PROGRAM IO_Mapping
VAR
	BLINK_500msOn_500MsOff	: Blink;
END_VAR

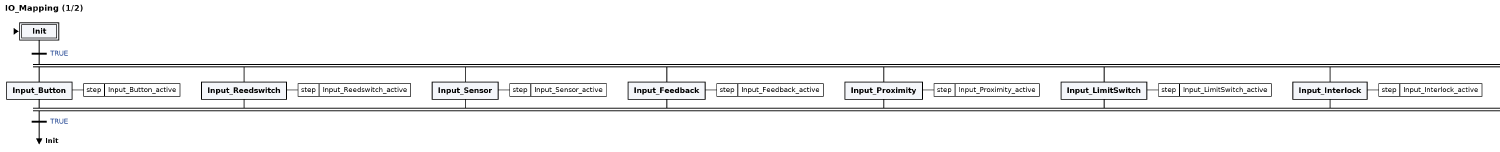
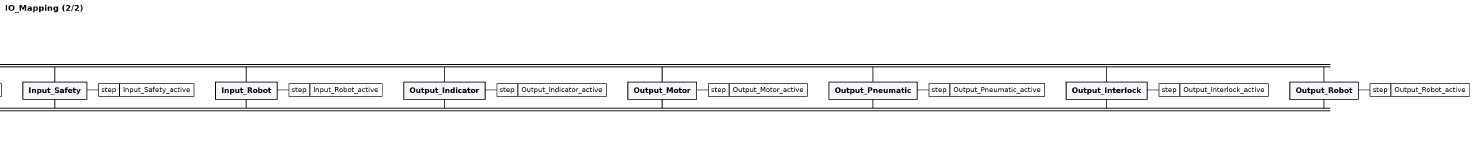
INITIAL_STEP Init:
END_STEP
TRANSITION FROM Init TO (Input_Button, Input_Reedswitch, Input_Sensor, Input_Feedback, Input_Proximity, Input_LimitSwitch, Input_Interlock, Input_Safety, Input_Robot, Output_Indicator, Output_Motor, Output_Pneumatic, Output_Interlock, Output_Robot)
    := TRUE;
END_TRANSITION
STEP Input_Button:
    Input_Button_active(N);  // step action
END_STEP
STEP Input_Reedswitch:
    Input_Reedswitch_active(N);  // step action
END_STEP
STEP Input_Sensor:
    Input_Sensor_active(N);  // step action
END_STEP
STEP Input_Feedback:
    Input_Feedback_active(N);  // step action
END_STEP
STEP Input_Proximity:
    Input_Proximity_active(N);  // step action
END_STEP
STEP Input_LimitSwitch:
    Input_LimitSwitch_active(N);  // step action
END_STEP
STEP Input_Interlock:
    Input_Interlock_active(N);  // step action
END_STEP
STEP Input_Safety:
    Input_Safety_active(N);  // step action
END_STEP
STEP Input_Robot:
    Input_Robot_active(N);  // step action
END_STEP
STEP Output_Indicator:
    Output_Indicator_active(N);  // step action
END_STEP
STEP Output_Motor:
    Output_Motor_active(N);  // step action
END_STEP
STEP Output_Pneumatic:
    Output_Pneumatic_active(N);  // step action
END_STEP
STEP Output_Interlock:
    Output_Interlock_active(N);  // step action
END_STEP
STEP Output_Robot:
    Output_Robot_active(N);  // step action
END_STEP
TRANSITION FROM (Input_Button, Input_Reedswitch, Input_Sensor, Input_Feedback, Input_Proximity, Input_LimitSwitch, Input_Interlock, Input_Safety, Input_Robot, Output_Indicator, Output_Motor, Output_Pneumatic, Output_Interlock, Output_Robot) TO Init
    := TRUE;
END_TRANSITION

ACTION Input_Button_active:
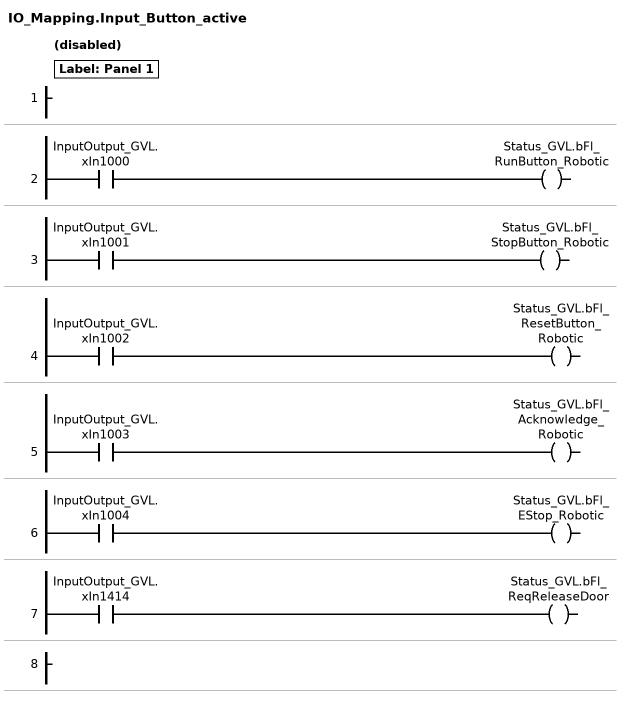
// NETWORK 1 (disabled)
// label: Label: Panel 1

// NETWORK 2
Status_GVL.bFl_RunButton_Robotic := InputOutput_GVL.xIn1000;

// NETWORK 3
Status_GVL.bFl_StopButton_Robotic := InputOutput_GVL.xIn1001;

// NETWORK 4
Status_GVL.bFl_ResetButton_Robotic := InputOutput_GVL.xIn1002;

// NETWORK 5
Status_GVL.bFl_Acknowledge_Robotic := InputOutput_GVL.xIn1003;

// NETWORK 6
Status_GVL.bFl_EStop_Robotic := InputOutput_GVL.xIn1004;

// NETWORK 7
Status_GVL.bFl_ReqReleaseDoor := InputOutput_GVL.xIn1414;

// NETWORK 8
END_ACTION

ACTION Input_Feedback_active:
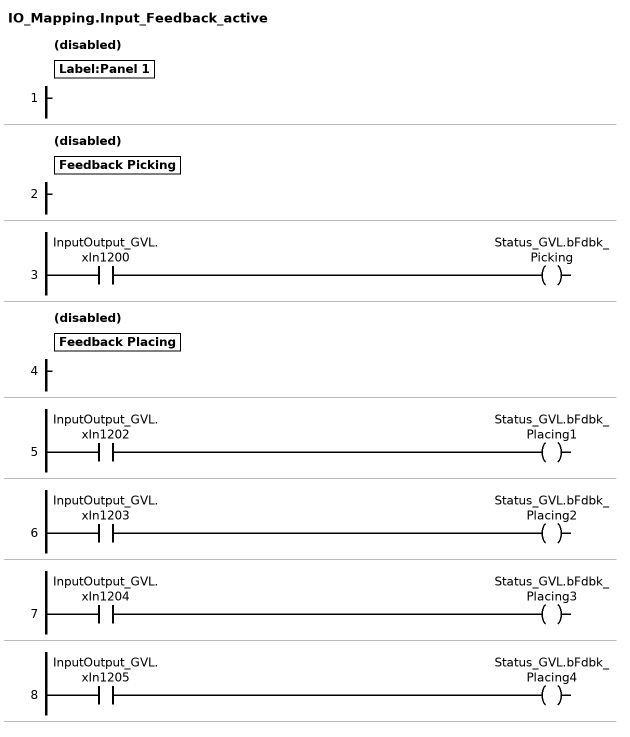
// NETWORK 1 (disabled)
// label: Label:Panel 1

// NETWORK 2 (disabled)
// label: Feedback Picking

// NETWORK 3
Status_GVL.bFdbk_Picking := InputOutput_GVL.xIn1200;

// NETWORK 4 (disabled)
// label: Feedback Placing

// NETWORK 5
Status_GVL.bFdbk_Placing1 := InputOutput_GVL.xIn1202;

// NETWORK 6
Status_GVL.bFdbk_Placing2 := InputOutput_GVL.xIn1203;

// NETWORK 7
Status_GVL.bFdbk_Placing3 := InputOutput_GVL.xIn1204;

// NETWORK 8
Status_GVL.bFdbk_Placing4 := InputOutput_GVL.xIn1205;
END_ACTION

ACTION Input_Interlock_active:
// NETWORK 1
END_ACTION

ACTION Input_LimitSwitch_active:
// NETWORK 1
END_ACTION

ACTION Input_Proximity_active:
// NETWORK 1 (disabled)
// label: Proximity

// NETWORK 2
END_ACTION

ACTION Input_Reedswitch_active:
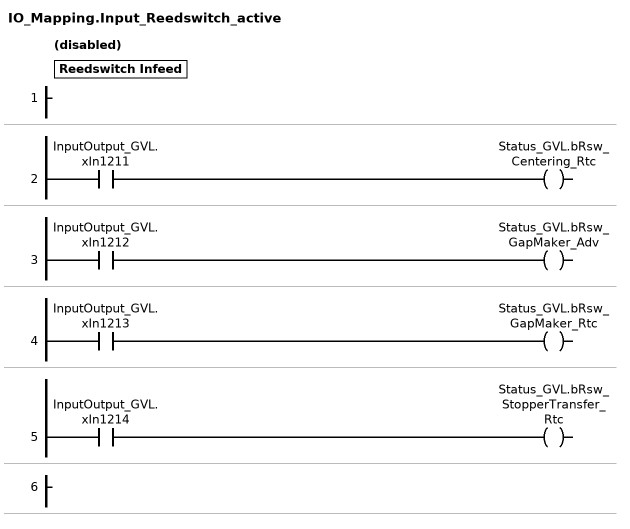
// NETWORK 1 (disabled)
// label: Reedswitch Infeed

// NETWORK 2
Status_GVL.bRsw_Centering_Rtc := InputOutput_GVL.xIn1211;

// NETWORK 3
Status_GVL.bRsw_GapMaker_Adv := InputOutput_GVL.xIn1212;

// NETWORK 4
Status_GVL.bRsw_GapMaker_Rtc := InputOutput_GVL.xIn1213;

// NETWORK 5
Status_GVL.bRsw_StopperTransfer_Rtc := InputOutput_GVL.xIn1214;

// NETWORK 6
END_ACTION

ACTION Input_Robot_active:
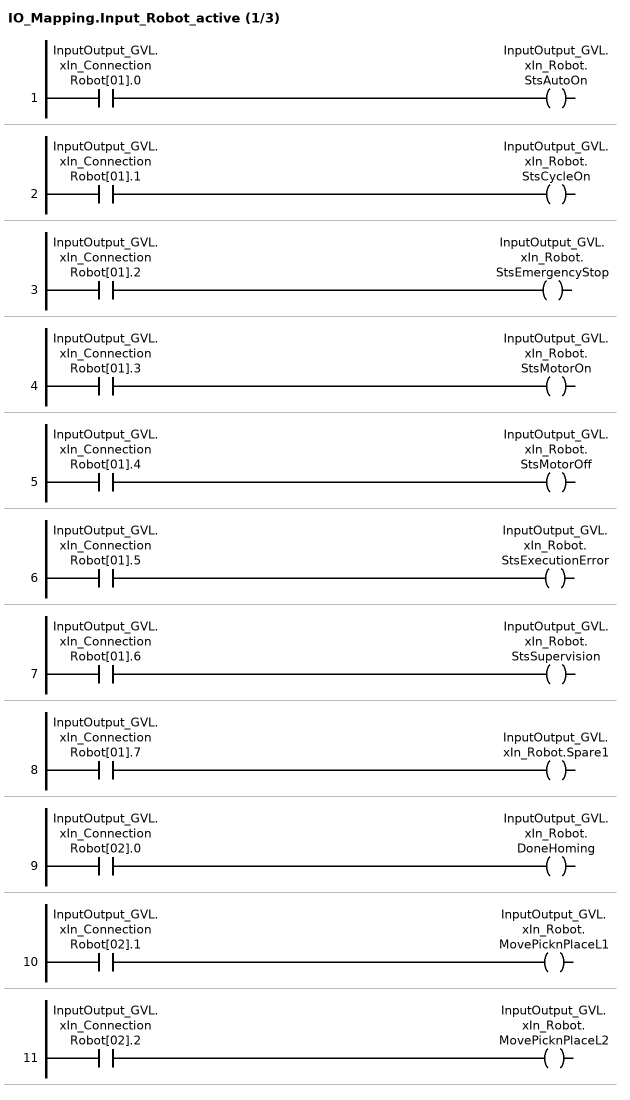
// NETWORK 1
InputOutput_GVL.xIn_Robot.StsAutoOn := InputOutput_GVL.xIn_ConnectionRobot[01].0;

// NETWORK 2
InputOutput_GVL.xIn_Robot.StsCycleOn := InputOutput_GVL.xIn_ConnectionRobot[01].1;

// NETWORK 3
InputOutput_GVL.xIn_Robot.StsEmergencyStop := InputOutput_GVL.xIn_ConnectionRobot[01].2;

// NETWORK 4
InputOutput_GVL.xIn_Robot.StsMotorOn := InputOutput_GVL.xIn_ConnectionRobot[01].3;

// NETWORK 5
InputOutput_GVL.xIn_Robot.StsMotorOff := InputOutput_GVL.xIn_ConnectionRobot[01].4;

// NETWORK 6
InputOutput_GVL.xIn_Robot.StsExecutionError := InputOutput_GVL.xIn_ConnectionRobot[01].5;

// NETWORK 7
InputOutput_GVL.xIn_Robot.StsSupervision := InputOutput_GVL.xIn_ConnectionRobot[01].6;

// NETWORK 8
InputOutput_GVL.xIn_Robot.Spare1 := InputOutput_GVL.xIn_ConnectionRobot[01].7;

// NETWORK 9
InputOutput_GVL.xIn_Robot.DoneHoming := InputOutput_GVL.xIn_ConnectionRobot[02].0;

// NETWORK 10
InputOutput_GVL.xIn_Robot.MovePicknPlaceL1 := InputOutput_GVL.xIn_ConnectionRobot[02].1;

// NETWORK 11
InputOutput_GVL.xIn_Robot.MovePicknPlaceL2 := InputOutput_GVL.xIn_ConnectionRobot[02].2;

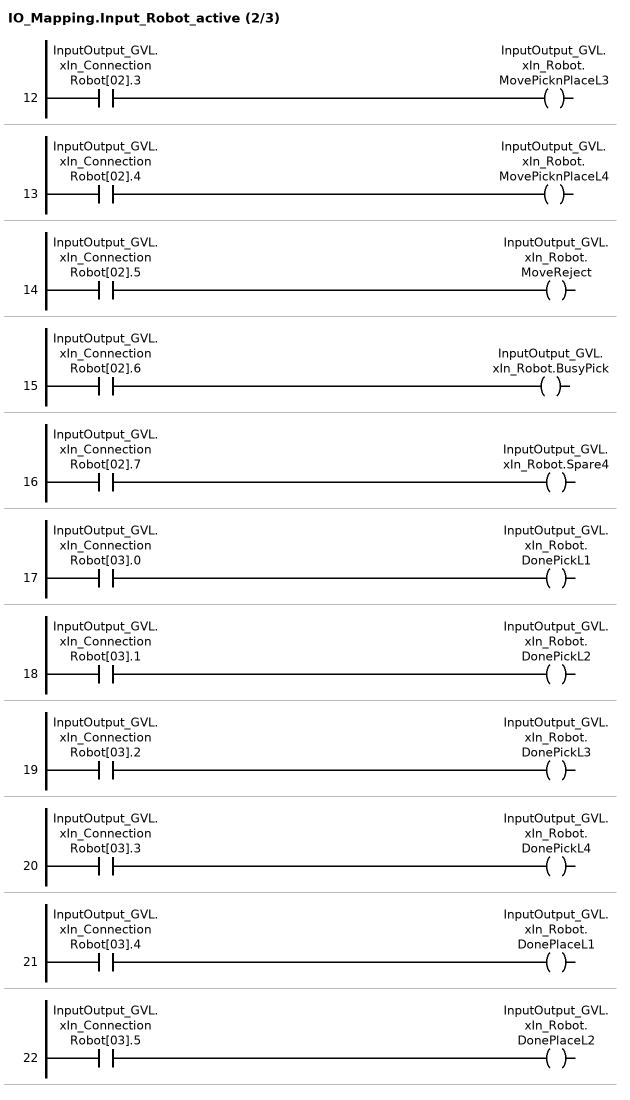
// NETWORK 12
InputOutput_GVL.xIn_Robot.MovePicknPlaceL3 := InputOutput_GVL.xIn_ConnectionRobot[02].3;

// NETWORK 13
InputOutput_GVL.xIn_Robot.MovePicknPlaceL4 := InputOutput_GVL.xIn_ConnectionRobot[02].4;

// NETWORK 14
InputOutput_GVL.xIn_Robot.MoveReject := InputOutput_GVL.xIn_ConnectionRobot[02].5;

// NETWORK 15
InputOutput_GVL.xIn_Robot.BusyPick := InputOutput_GVL.xIn_ConnectionRobot[02].6;

// NETWORK 16
InputOutput_GVL.xIn_Robot.Spare4 := InputOutput_GVL.xIn_ConnectionRobot[02].7;

// NETWORK 17
InputOutput_GVL.xIn_Robot.DonePickL1 := InputOutput_GVL.xIn_ConnectionRobot[03].0;

// NETWORK 18
InputOutput_GVL.xIn_Robot.DonePickL2 := InputOutput_GVL.xIn_ConnectionRobot[03].1;

// NETWORK 19
InputOutput_GVL.xIn_Robot.DonePickL3 := InputOutput_GVL.xIn_ConnectionRobot[03].2;

// NETWORK 20
InputOutput_GVL.xIn_Robot.DonePickL4 := InputOutput_GVL.xIn_ConnectionRobot[03].3;

// NETWORK 21
InputOutput_GVL.xIn_Robot.DonePlaceL1 := InputOutput_GVL.xIn_ConnectionRobot[03].4;

// NETWORK 22
InputOutput_GVL.xIn_Robot.DonePlaceL2 := InputOutput_GVL.xIn_ConnectionRobot[03].5;

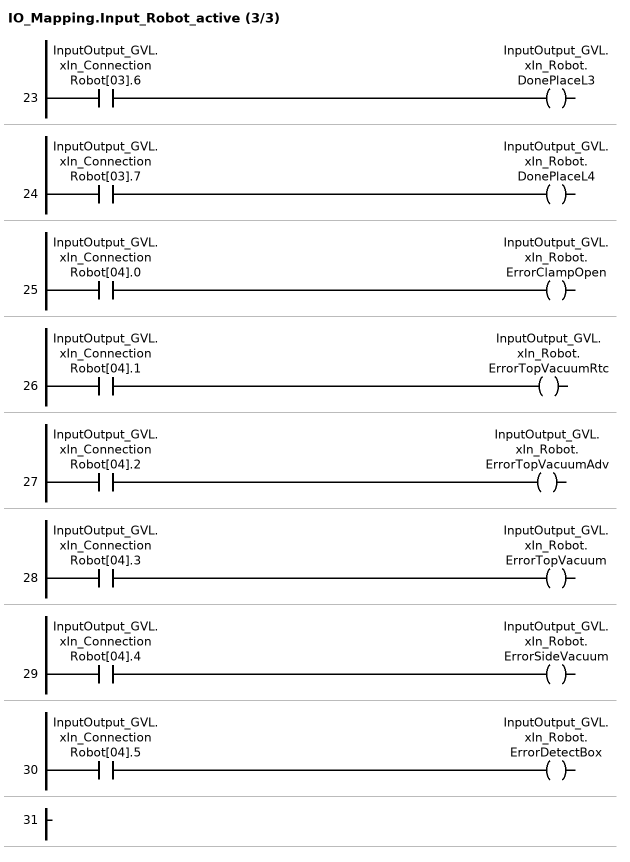
// NETWORK 23
InputOutput_GVL.xIn_Robot.DonePlaceL3 := InputOutput_GVL.xIn_ConnectionRobot[03].6;

// NETWORK 24
InputOutput_GVL.xIn_Robot.DonePlaceL4 := InputOutput_GVL.xIn_ConnectionRobot[03].7;

// NETWORK 25
InputOutput_GVL.xIn_Robot.ErrorClampOpen := InputOutput_GVL.xIn_ConnectionRobot[04].0;

// NETWORK 26
InputOutput_GVL.xIn_Robot.ErrorTopVacuumRtc := InputOutput_GVL.xIn_ConnectionRobot[04].1;

// NETWORK 27
InputOutput_GVL.xIn_Robot.ErrorTopVacuumAdv := InputOutput_GVL.xIn_ConnectionRobot[04].2;

// NETWORK 28
InputOutput_GVL.xIn_Robot.ErrorTopVacuum := InputOutput_GVL.xIn_ConnectionRobot[04].3;

// NETWORK 29
InputOutput_GVL.xIn_Robot.ErrorSideVacuum := InputOutput_GVL.xIn_ConnectionRobot[04].4;

// NETWORK 30
InputOutput_GVL.xIn_Robot.ErrorDetectBox := InputOutput_GVL.xIn_ConnectionRobot[04].5;

// NETWORK 31
END_ACTION

ACTION Input_Safety_active:
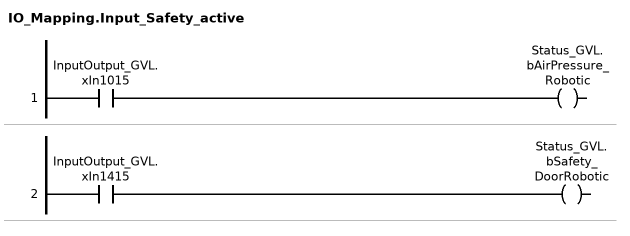
// NETWORK 1
Status_GVL.bAirPressure_Robotic := InputOutput_GVL.xIn1015;

// NETWORK 2
Status_GVL.bSafety_DoorRobotic := InputOutput_GVL.xIn1415;
END_ACTION

ACTION Input_Sensor_active:
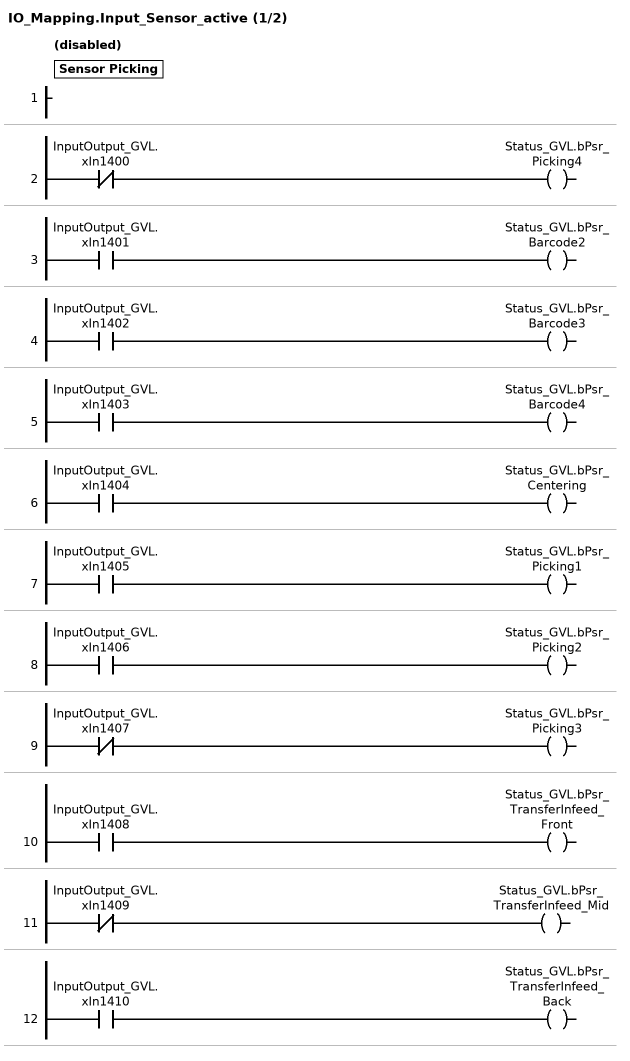
// NETWORK 1 (disabled)
// label: Sensor Picking

// NETWORK 2
Status_GVL.bPsr_Picking4 := NOT InputOutput_GVL.xIn1400;

// NETWORK 3
Status_GVL.bPsr_Barcode2 := InputOutput_GVL.xIn1401;

// NETWORK 4
Status_GVL.bPsr_Barcode3 := InputOutput_GVL.xIn1402;

// NETWORK 5
Status_GVL.bPsr_Barcode4 := InputOutput_GVL.xIn1403;

// NETWORK 6
Status_GVL.bPsr_Centering := InputOutput_GVL.xIn1404;

// NETWORK 7
Status_GVL.bPsr_Picking1 := InputOutput_GVL.xIn1405;

// NETWORK 8
Status_GVL.bPsr_Picking2 := InputOutput_GVL.xIn1406;

// NETWORK 9
Status_GVL.bPsr_Picking3 := NOT InputOutput_GVL.xIn1407;

// NETWORK 10
Status_GVL.bPsr_TransferInfeed_Front := InputOutput_GVL.xIn1408;

// NETWORK 11
Status_GVL.bPsr_TransferInfeed_Mid := NOT InputOutput_GVL.xIn1409;

// NETWORK 12
Status_GVL.bPsr_TransferInfeed_Back := InputOutput_GVL.xIn1410;

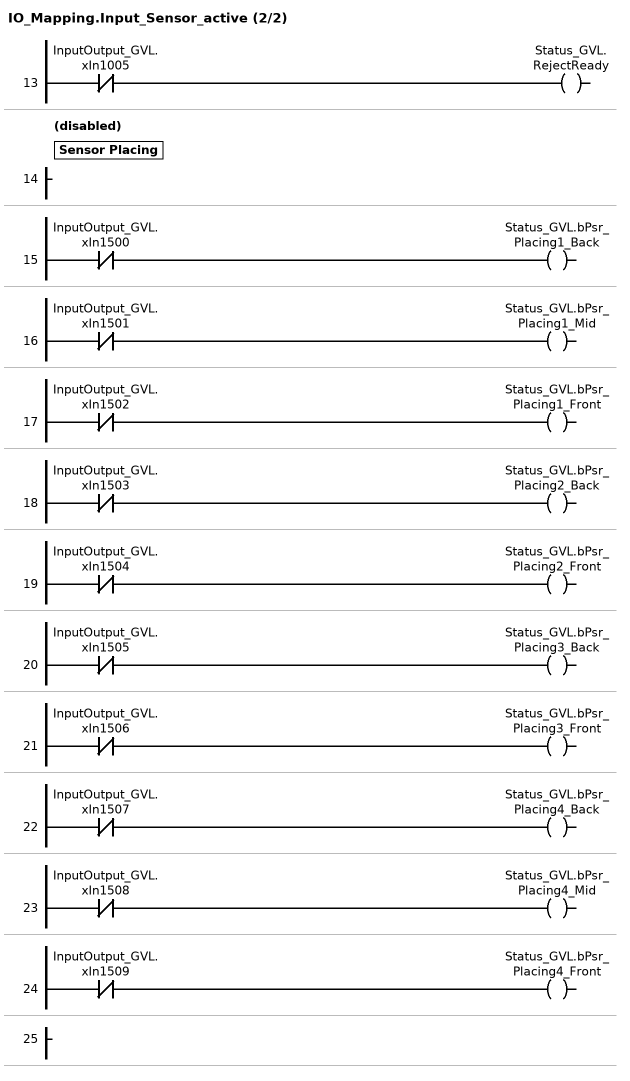
// NETWORK 13
Status_GVL.RejectReady := NOT InputOutput_GVL.xIn1005;

// NETWORK 14 (disabled)
// label: Sensor Placing

// NETWORK 15
Status_GVL.bPsr_Placing1_Back := NOT InputOutput_GVL.xIn1500;

// NETWORK 16
Status_GVL.bPsr_Placing1_Mid := NOT InputOutput_GVL.xIn1501;

// NETWORK 17
Status_GVL.bPsr_Placing1_Front := NOT InputOutput_GVL.xIn1502;

// NETWORK 18
Status_GVL.bPsr_Placing2_Back := NOT InputOutput_GVL.xIn1503;

// NETWORK 19
Status_GVL.bPsr_Placing2_Front := NOT InputOutput_GVL.xIn1504;

// NETWORK 20
Status_GVL.bPsr_Placing3_Back := NOT InputOutput_GVL.xIn1505;

// NETWORK 21
Status_GVL.bPsr_Placing3_Front := NOT InputOutput_GVL.xIn1506;

// NETWORK 22
Status_GVL.bPsr_Placing4_Back := NOT InputOutput_GVL.xIn1507;

// NETWORK 23
Status_GVL.bPsr_Placing4_Mid := NOT InputOutput_GVL.xIn1508;

// NETWORK 24
Status_GVL.bPsr_Placing4_Front := NOT InputOutput_GVL.xIn1509;

// NETWORK 25
END_ACTION

ACTION Output_Indicator_active:
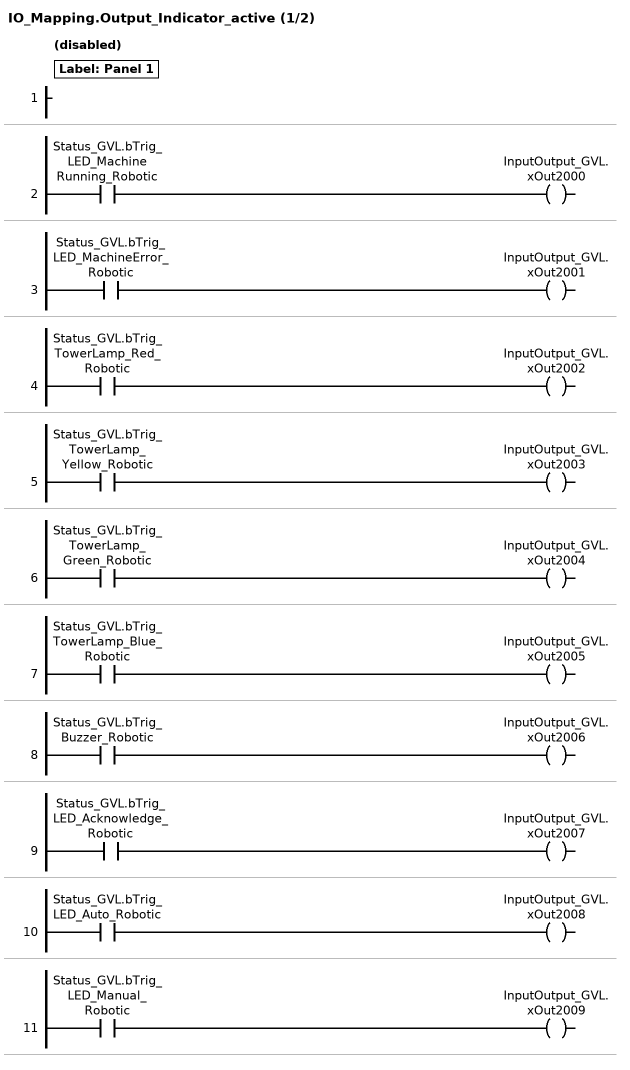
// NETWORK 1 (disabled)
// label: Label: Panel 1

// NETWORK 2
InputOutput_GVL.xOut2000 := Status_GVL.bTrig_LED_MachineRunning_Robotic;

// NETWORK 3
InputOutput_GVL.xOut2001 := Status_GVL.bTrig_LED_MachineError_Robotic;

// NETWORK 4
InputOutput_GVL.xOut2002 := Status_GVL.bTrig_TowerLamp_Red_Robotic;

// NETWORK 5
InputOutput_GVL.xOut2003 := Status_GVL.bTrig_TowerLamp_Yellow_Robotic;

// NETWORK 6
InputOutput_GVL.xOut2004 := Status_GVL.bTrig_TowerLamp_Green_Robotic;

// NETWORK 7
InputOutput_GVL.xOut2005 := Status_GVL.bTrig_TowerLamp_Blue_Robotic;

// NETWORK 8
InputOutput_GVL.xOut2006 := Status_GVL.bTrig_Buzzer_Robotic;

// NETWORK 9
InputOutput_GVL.xOut2007 := Status_GVL.bTrig_LED_Acknowledge_Robotic;

// NETWORK 10
InputOutput_GVL.xOut2008 := Status_GVL.bTrig_LED_Auto_Robotic;

// NETWORK 11
InputOutput_GVL.xOut2009 := Status_GVL.bTrig_LED_Manual_Robotic;

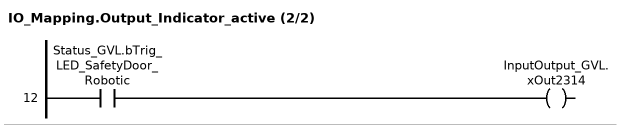
// NETWORK 12
InputOutput_GVL.xOut2314 := Status_GVL.bTrig_LED_SafetyDoor_Robotic;
END_ACTION

ACTION Output_Interlock_active:
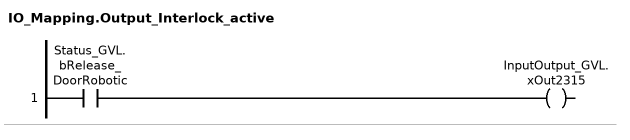
// NETWORK 1
InputOutput_GVL.xOut2315 := Status_GVL.bRelease_DoorRobotic;
END_ACTION

ACTION Output_Motor_active:
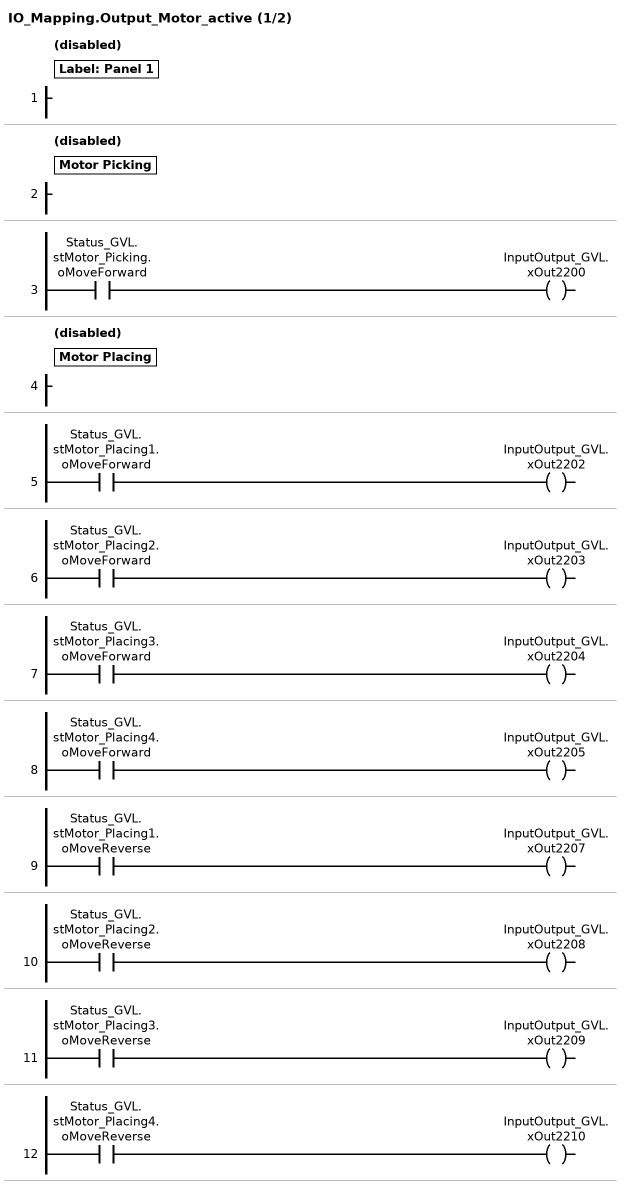
// NETWORK 1 (disabled)
// label: Label: Panel 1

// NETWORK 2 (disabled)
// label: Motor Picking

// NETWORK 3
InputOutput_GVL.xOut2200 := Status_GVL.stMotor_Picking.oMoveForward;

// NETWORK 4 (disabled)
// label: Motor Placing

// NETWORK 5
InputOutput_GVL.xOut2202 := Status_GVL.stMotor_Placing1.oMoveForward;

// NETWORK 6
InputOutput_GVL.xOut2203 := Status_GVL.stMotor_Placing2.oMoveForward;

// NETWORK 7
InputOutput_GVL.xOut2204 := Status_GVL.stMotor_Placing3.oMoveForward;

// NETWORK 8
InputOutput_GVL.xOut2205 := Status_GVL.stMotor_Placing4.oMoveForward;

// NETWORK 9
InputOutput_GVL.xOut2207 := Status_GVL.stMotor_Placing1.oMoveReverse;

// NETWORK 10
InputOutput_GVL.xOut2208 := Status_GVL.stMotor_Placing2.oMoveReverse;

// NETWORK 11
InputOutput_GVL.xOut2209 := Status_GVL.stMotor_Placing3.oMoveReverse;

// NETWORK 12
InputOutput_GVL.xOut2210 := Status_GVL.stMotor_Placing4.oMoveReverse;

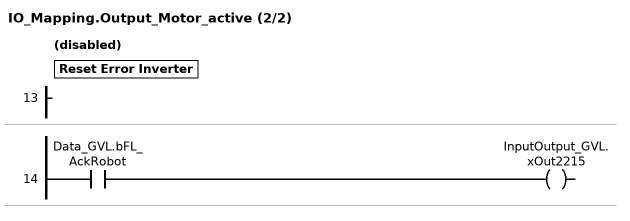
// NETWORK 13 (disabled)
// label: Reset Error Inverter

// NETWORK 14
InputOutput_GVL.xOut2215 := Data_GVL.bFL_AckRobot;
END_ACTION

ACTION Output_Pneumatic_active:
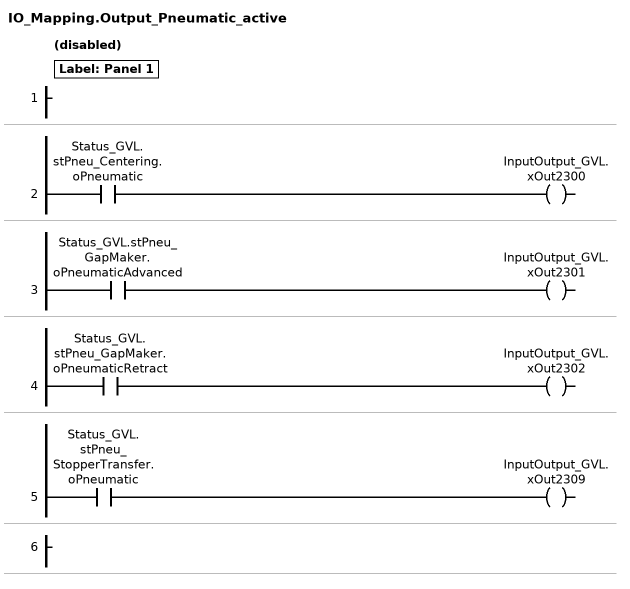
// NETWORK 1 (disabled)
// label: Label: Panel 1

// NETWORK 2
InputOutput_GVL.xOut2300 := Status_GVL.stPneu_Centering.oPneumatic;

// NETWORK 3
InputOutput_GVL.xOut2301 := Status_GVL.stPneu_GapMaker.oPneumaticAdvanced;

// NETWORK 4
InputOutput_GVL.xOut2302 := Status_GVL.stPneu_GapMaker.oPneumaticRetract;

// NETWORK 5
InputOutput_GVL.xOut2309 := Status_GVL.stPneu_StopperTransfer.oPneumatic;

// NETWORK 6
END_ACTION

ACTION Output_Robot_active:
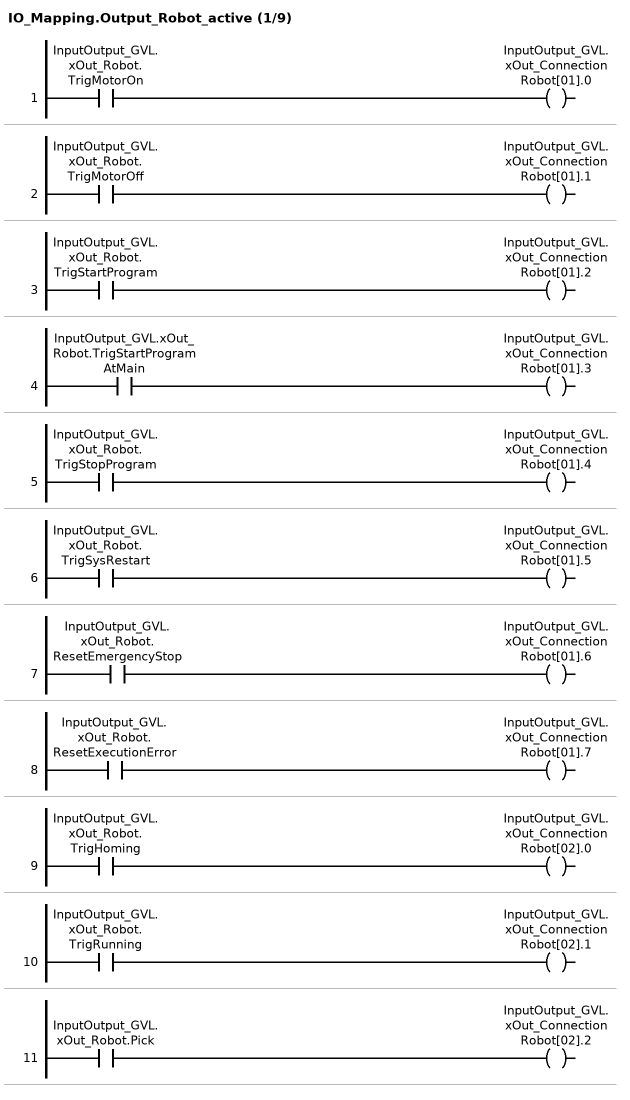
// NETWORK 1
InputOutput_GVL.xOut_ConnectionRobot[01].0 := InputOutput_GVL.xOut_Robot.TrigMotorOn;

// NETWORK 2
InputOutput_GVL.xOut_ConnectionRobot[01].1 := InputOutput_GVL.xOut_Robot.TrigMotorOff;

// NETWORK 3
InputOutput_GVL.xOut_ConnectionRobot[01].2 := InputOutput_GVL.xOut_Robot.TrigStartProgram;

// NETWORK 4
InputOutput_GVL.xOut_ConnectionRobot[01].3 := InputOutput_GVL.xOut_Robot.TrigStartProgramAtMain;

// NETWORK 5
InputOutput_GVL.xOut_ConnectionRobot[01].4 := InputOutput_GVL.xOut_Robot.TrigStopProgram;

// NETWORK 6
InputOutput_GVL.xOut_ConnectionRobot[01].5 := InputOutput_GVL.xOut_Robot.TrigSysRestart;

// NETWORK 7
InputOutput_GVL.xOut_ConnectionRobot[01].6 := InputOutput_GVL.xOut_Robot.ResetEmergencyStop;

// NETWORK 8
InputOutput_GVL.xOut_ConnectionRobot[01].7 := InputOutput_GVL.xOut_Robot.ResetExecutionError;

// NETWORK 9
InputOutput_GVL.xOut_ConnectionRobot[02].0 := InputOutput_GVL.xOut_Robot.TrigHoming;

// NETWORK 10
InputOutput_GVL.xOut_ConnectionRobot[02].1 := InputOutput_GVL.xOut_Robot.TrigRunning;

// NETWORK 11
InputOutput_GVL.xOut_ConnectionRobot[02].2 := InputOutput_GVL.xOut_Robot.Pick;

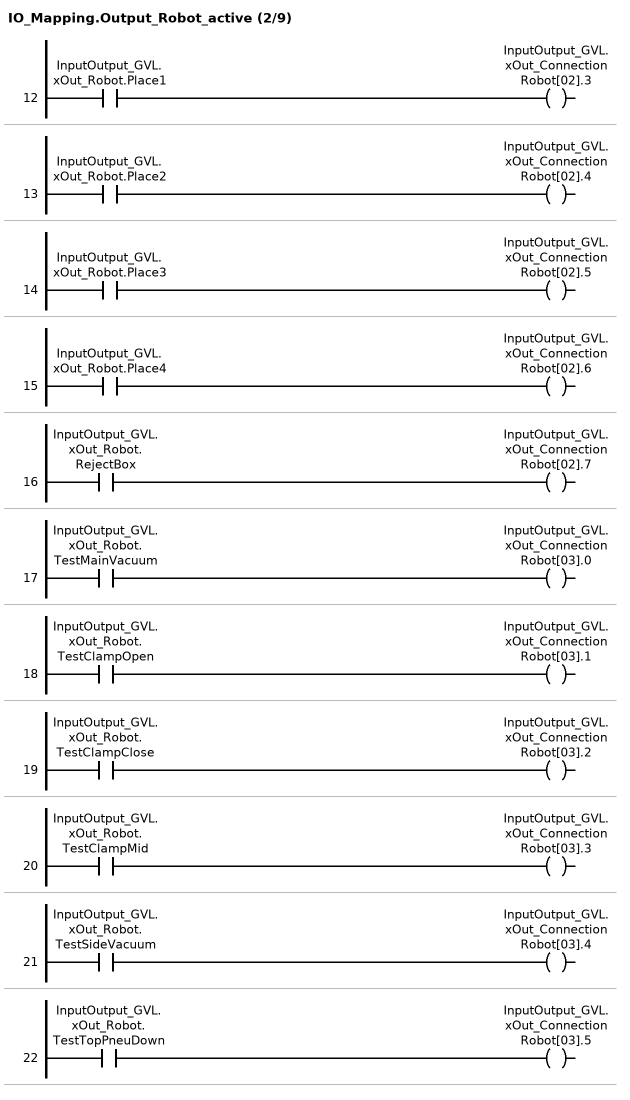
// NETWORK 12
InputOutput_GVL.xOut_ConnectionRobot[02].3 := InputOutput_GVL.xOut_Robot.Place1;

// NETWORK 13
InputOutput_GVL.xOut_ConnectionRobot[02].4 := InputOutput_GVL.xOut_Robot.Place2;

// NETWORK 14
InputOutput_GVL.xOut_ConnectionRobot[02].5 := InputOutput_GVL.xOut_Robot.Place3;

// NETWORK 15
InputOutput_GVL.xOut_ConnectionRobot[02].6 := InputOutput_GVL.xOut_Robot.Place4;

// NETWORK 16
InputOutput_GVL.xOut_ConnectionRobot[02].7 := InputOutput_GVL.xOut_Robot.RejectBox;

// NETWORK 17
InputOutput_GVL.xOut_ConnectionRobot[03].0 := InputOutput_GVL.xOut_Robot.TestMainVacuum;

// NETWORK 18
InputOutput_GVL.xOut_ConnectionRobot[03].1 := InputOutput_GVL.xOut_Robot.TestClampOpen;

// NETWORK 19
InputOutput_GVL.xOut_ConnectionRobot[03].2 := InputOutput_GVL.xOut_Robot.TestClampClose;

// NETWORK 20
InputOutput_GVL.xOut_ConnectionRobot[03].3 := InputOutput_GVL.xOut_Robot.TestClampMid;

// NETWORK 21
InputOutput_GVL.xOut_ConnectionRobot[03].4 := InputOutput_GVL.xOut_Robot.TestSideVacuum;

// NETWORK 22
InputOutput_GVL.xOut_ConnectionRobot[03].5 := InputOutput_GVL.xOut_Robot.TestTopPneuDown;

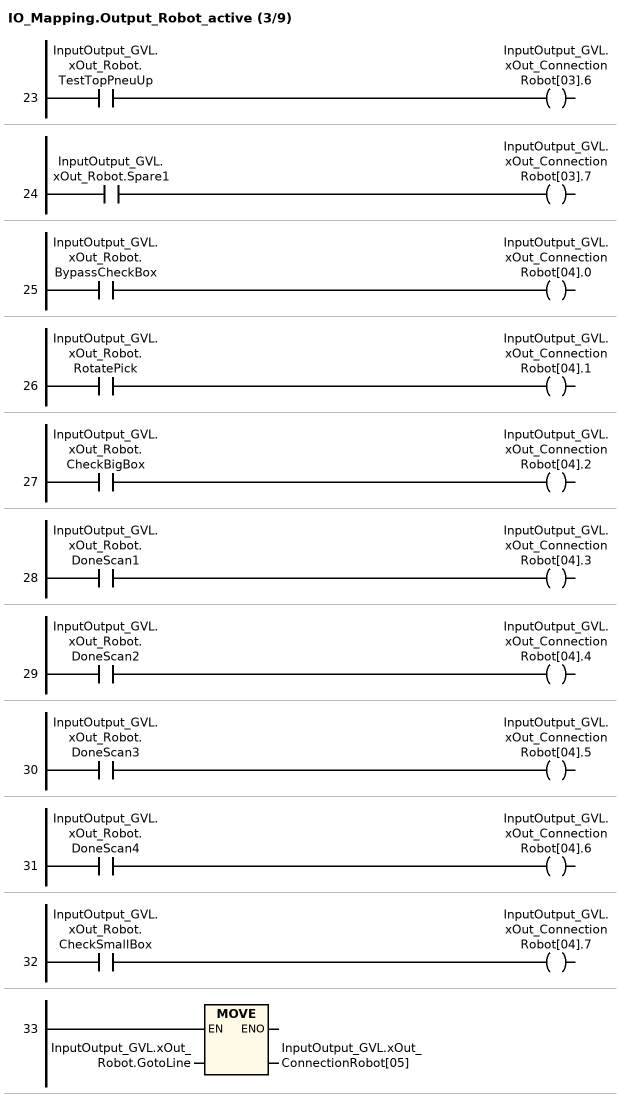
// NETWORK 23
InputOutput_GVL.xOut_ConnectionRobot[03].6 := InputOutput_GVL.xOut_Robot.TestTopPneuUp;

// NETWORK 24
InputOutput_GVL.xOut_ConnectionRobot[03].7 := InputOutput_GVL.xOut_Robot.Spare1;

// NETWORK 25
InputOutput_GVL.xOut_ConnectionRobot[04].0 := InputOutput_GVL.xOut_Robot.BypassCheckBox;

// NETWORK 26
InputOutput_GVL.xOut_ConnectionRobot[04].1 := InputOutput_GVL.xOut_Robot.RotatePick;

// NETWORK 27
InputOutput_GVL.xOut_ConnectionRobot[04].2 := InputOutput_GVL.xOut_Robot.CheckBigBox;

// NETWORK 28
InputOutput_GVL.xOut_ConnectionRobot[04].3 := InputOutput_GVL.xOut_Robot.DoneScan1;

// NETWORK 29
InputOutput_GVL.xOut_ConnectionRobot[04].4 := InputOutput_GVL.xOut_Robot.DoneScan2;

// NETWORK 30
InputOutput_GVL.xOut_ConnectionRobot[04].5 := InputOutput_GVL.xOut_Robot.DoneScan3;

// NETWORK 31
InputOutput_GVL.xOut_ConnectionRobot[04].6 := InputOutput_GVL.xOut_Robot.DoneScan4;

// NETWORK 32
InputOutput_GVL.xOut_ConnectionRobot[04].7 := InputOutput_GVL.xOut_Robot.CheckSmallBox;

// NETWORK 33
InputOutput_GVL.xOut_ConnectionRobot[05] := InputOutput_GVL.xOut_Robot.GotoLine;

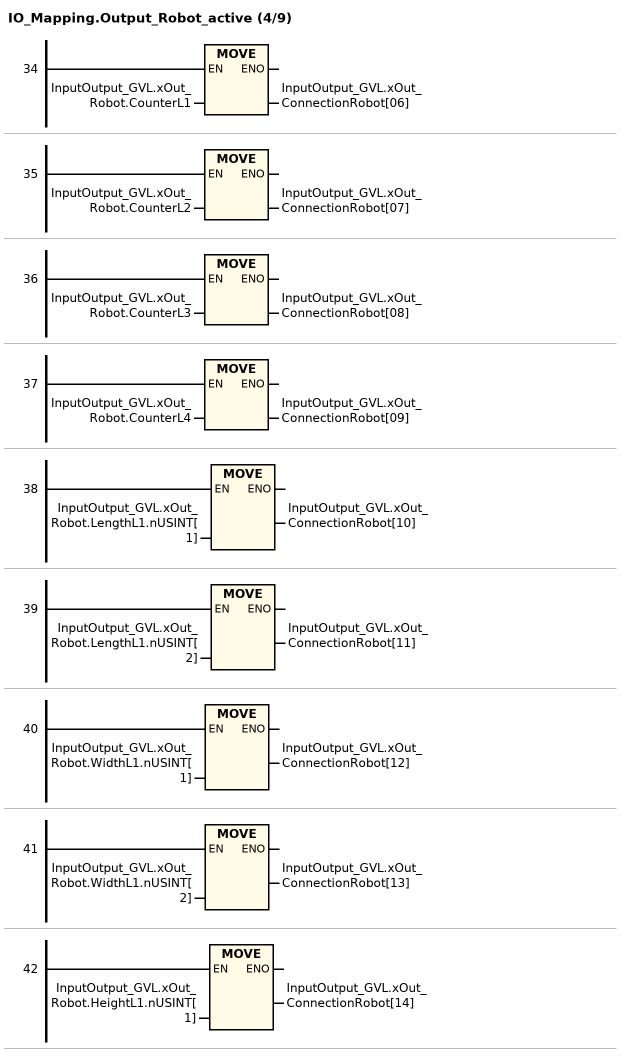
// NETWORK 34
InputOutput_GVL.xOut_ConnectionRobot[06] := InputOutput_GVL.xOut_Robot.CounterL1;

// NETWORK 35
InputOutput_GVL.xOut_ConnectionRobot[07] := InputOutput_GVL.xOut_Robot.CounterL2;

// NETWORK 36
InputOutput_GVL.xOut_ConnectionRobot[08] := InputOutput_GVL.xOut_Robot.CounterL3;

// NETWORK 37
InputOutput_GVL.xOut_ConnectionRobot[09] := InputOutput_GVL.xOut_Robot.CounterL4;

// NETWORK 38
InputOutput_GVL.xOut_ConnectionRobot[10] := InputOutput_GVL.xOut_Robot.LengthL1.nUSINT[1];

// NETWORK 39
InputOutput_GVL.xOut_ConnectionRobot[11] := InputOutput_GVL.xOut_Robot.LengthL1.nUSINT[2];

// NETWORK 40
InputOutput_GVL.xOut_ConnectionRobot[12] := InputOutput_GVL.xOut_Robot.WidthL1.nUSINT[1];

// NETWORK 41
InputOutput_GVL.xOut_ConnectionRobot[13] := InputOutput_GVL.xOut_Robot.WidthL1.nUSINT[2];

// NETWORK 42
InputOutput_GVL.xOut_ConnectionRobot[14] := InputOutput_GVL.xOut_Robot.HeightL1.nUSINT[1];

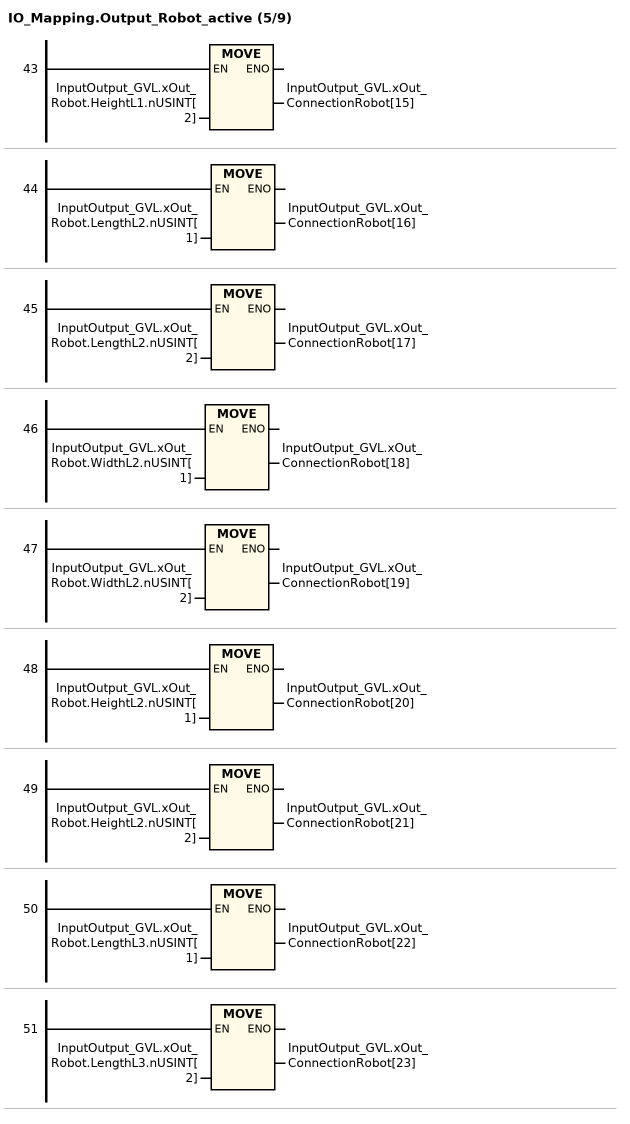
// NETWORK 43
InputOutput_GVL.xOut_ConnectionRobot[15] := InputOutput_GVL.xOut_Robot.HeightL1.nUSINT[2];

// NETWORK 44
InputOutput_GVL.xOut_ConnectionRobot[16] := InputOutput_GVL.xOut_Robot.LengthL2.nUSINT[1];

// NETWORK 45
InputOutput_GVL.xOut_ConnectionRobot[17] := InputOutput_GVL.xOut_Robot.LengthL2.nUSINT[2];

// NETWORK 46
InputOutput_GVL.xOut_ConnectionRobot[18] := InputOutput_GVL.xOut_Robot.WidthL2.nUSINT[1];

// NETWORK 47
InputOutput_GVL.xOut_ConnectionRobot[19] := InputOutput_GVL.xOut_Robot.WidthL2.nUSINT[2];

// NETWORK 48
InputOutput_GVL.xOut_ConnectionRobot[20] := InputOutput_GVL.xOut_Robot.HeightL2.nUSINT[1];

// NETWORK 49
InputOutput_GVL.xOut_ConnectionRobot[21] := InputOutput_GVL.xOut_Robot.HeightL2.nUSINT[2];

// NETWORK 50
InputOutput_GVL.xOut_ConnectionRobot[22] := InputOutput_GVL.xOut_Robot.LengthL3.nUSINT[1];

// NETWORK 51
InputOutput_GVL.xOut_ConnectionRobot[23] := InputOutput_GVL.xOut_Robot.LengthL3.nUSINT[2];

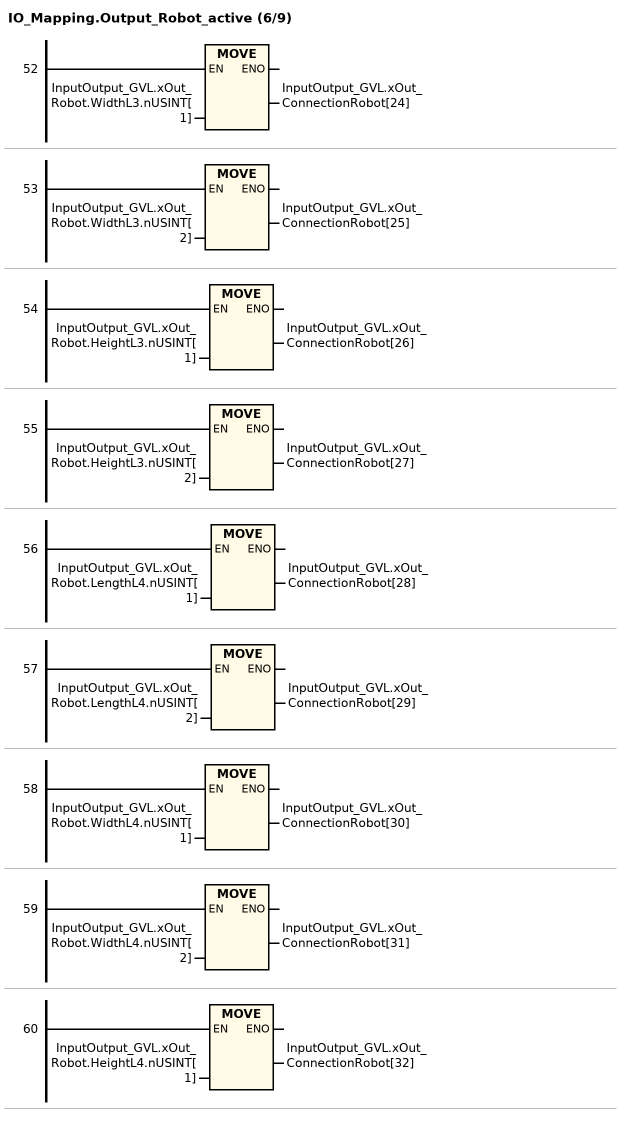
// NETWORK 52
InputOutput_GVL.xOut_ConnectionRobot[24] := InputOutput_GVL.xOut_Robot.WidthL3.nUSINT[1];

// NETWORK 53
InputOutput_GVL.xOut_ConnectionRobot[25] := InputOutput_GVL.xOut_Robot.WidthL3.nUSINT[2];

// NETWORK 54
InputOutput_GVL.xOut_ConnectionRobot[26] := InputOutput_GVL.xOut_Robot.HeightL3.nUSINT[1];

// NETWORK 55
InputOutput_GVL.xOut_ConnectionRobot[27] := InputOutput_GVL.xOut_Robot.HeightL3.nUSINT[2];

// NETWORK 56
InputOutput_GVL.xOut_ConnectionRobot[28] := InputOutput_GVL.xOut_Robot.LengthL4.nUSINT[1];

// NETWORK 57
InputOutput_GVL.xOut_ConnectionRobot[29] := InputOutput_GVL.xOut_Robot.LengthL4.nUSINT[2];

// NETWORK 58
InputOutput_GVL.xOut_ConnectionRobot[30] := InputOutput_GVL.xOut_Robot.WidthL4.nUSINT[1];

// NETWORK 59
InputOutput_GVL.xOut_ConnectionRobot[31] := InputOutput_GVL.xOut_Robot.WidthL4.nUSINT[2];

// NETWORK 60
InputOutput_GVL.xOut_ConnectionRobot[32] := InputOutput_GVL.xOut_Robot.HeightL4.nUSINT[1];

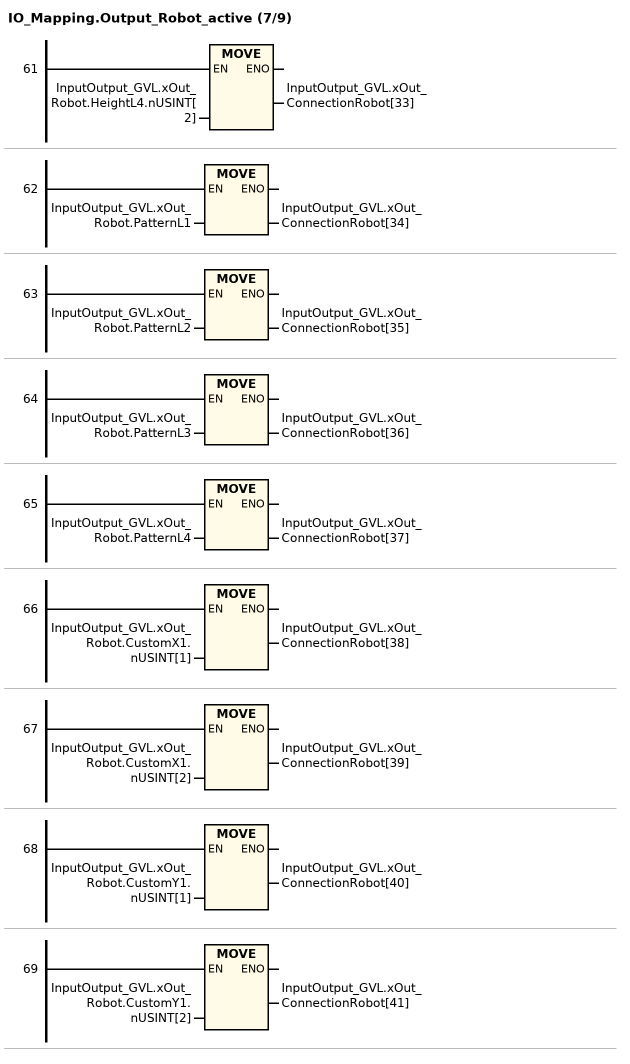
// NETWORK 61
InputOutput_GVL.xOut_ConnectionRobot[33] := InputOutput_GVL.xOut_Robot.HeightL4.nUSINT[2];

// NETWORK 62
InputOutput_GVL.xOut_ConnectionRobot[34] := InputOutput_GVL.xOut_Robot.PatternL1;

// NETWORK 63
InputOutput_GVL.xOut_ConnectionRobot[35] := InputOutput_GVL.xOut_Robot.PatternL2;

// NETWORK 64
InputOutput_GVL.xOut_ConnectionRobot[36] := InputOutput_GVL.xOut_Robot.PatternL3;

// NETWORK 65
InputOutput_GVL.xOut_ConnectionRobot[37] := InputOutput_GVL.xOut_Robot.PatternL4;

// NETWORK 66
InputOutput_GVL.xOut_ConnectionRobot[38] := InputOutput_GVL.xOut_Robot.CustomX1.nUSINT[1];

// NETWORK 67
InputOutput_GVL.xOut_ConnectionRobot[39] := InputOutput_GVL.xOut_Robot.CustomX1.nUSINT[2];

// NETWORK 68
InputOutput_GVL.xOut_ConnectionRobot[40] := InputOutput_GVL.xOut_Robot.CustomY1.nUSINT[1];

// NETWORK 69
InputOutput_GVL.xOut_ConnectionRobot[41] := InputOutput_GVL.xOut_Robot.CustomY1.nUSINT[2];

